ABB RobotStudio station: Process_and_Safety_V2.rsstnx

Station Process_and_Safety_V2 (saved by RobotStudio 23.2.10395.0)
Controller CRB1100_4_47
  mechanical unit ROB_1: CRB1100_4_47__01, 6 joints, base frame (0, 0, 0) mm
Layout (positions relative to the parent item):
  - CRB1100_4_47__01 [mechanism, from %ABB.RobotStudio.Models.CRB1100%\CRB1100_4_47__01.rslib] at (0, 0, 0) mm; joint values [-0.1244, 0.7509, -0.641, 0, 1.4609, -1.6952] (rad or m)
  - My_Mechanism [mechanism] at (0, 0, 0) mm; joint values [0, 0] (rad or m)
      TCP My_Mechanism_1 at (0, 0, 110) mm
      links: L1, L2, L3
  - P001 - Magazine rings [part] at (0, 500, 3) mm, rotated rx 90 ry 0 rz 0 deg, size 68.8 x 79.8 x 194.8 mm
  - P002 - Magazine nuts [part] at (100, 500, 3) mm, rotated rx 90 ry 0 rz 0 deg, size 68.8 x 106.2 x 289.3 mm
  - P004 - Fixture valve body [part] at (400, -50, 19.5) mm, rotated rx 90 ry 0 rz 0 deg, size 55 x 29 x 55 mm
  - P006 - Magazine bodies [part] at (-250, -400, 0) mm, rotated rx 90 ry 0 rz 0 deg, size 68.8 x 305 x 69.5 mm
  - P006a - Magazine bodies support [part] at (-243.75, -400, 85.1) mm, rotated rx 90 ry 0 rz 0 deg, size 40 x 15 x 5 mm
  - P007 - Magazine big nut [part] at (-100, 500, 3) mm, rotated rx 90 ry 0 rz 0 deg, size 68.8 x 91 x 212.5 mm
  - P006a - Magazine bodies support_2 [part] at (-243.75, -400, 145.1) mm, rotated rx 90 ry 0 rz 0 deg, size 40 x 15 x 5 mm
  - P006a - Magazine bodies support_3 [part] at (-243.75, -400, 205.1) mm, rotated rx 90 ry 0 rz 0 deg, size 40 x 15 x 5 mm
  - P006a - Magazine bodies support_4 [part] at (-243.75, -400, 265.1) mm, rotated rx 90 ry 0 rz 0 deg, size 40 x 15 x 5 mm
  - P006a - Magazine bodies support_5 [part] at (-243.75, -400, 25.1) mm, rotated rx 90 ry 0 rz 0 deg, size 40 x 15 x 5 mm
  - A001 - Grijper_2 [part] at (0, 0, 30) mm, rotated rx -90 ry 0 rz 0 deg, size 42 x 60 x 33 mm
  - Part_5 [part] at (0, 0, 30) mm, rotated rx -90 ry 0 rz 0 deg, size 52 x 72 x 22.6 mm
  - Part_6 [part] at (0, 0, 30) mm, rotated rx -90 ry 0 rz 0 deg, size 52 x 72 x 22.6 mm
  - GripperV2 [mechanism] at (89.85, -63.01, 369.8) mm, rotated rx -172.85 ry 3.1 rz -46.9 deg; joint values [0.008, -0.008] (rad or m)
      TCP GripperV2_1 at (0, -80, 0) mm, rotated rx 90 ry 0 rz 0 deg
      links: L1, L2, L3
  - P005 - Grote moer [part] at (-100, 385.14, 20.17) mm, rotated rx 97.62 ry -12.95 rz 59.14 deg, size 34.6 x 16.1 x 30 mm
  - P002 - Moer [part] at (100, 383.67, 26.5) mm, rotated rx 101.36 ry -6.49 rz 29.35 deg, size 24 x 13.5 x 27.7 mm
  - P001 - Sluitring [part] at (0, 381.43, 22.9) mm, rotated rx 103.06 ry 0 rz 0 deg, size 17.4 x 7.9 x 17.5 mm
  - P003 - Verlengstuk [part] at (-203.75, -400, 267.1) mm, rotated rx 0 ry 0 rz 90 deg, size 23.7 x 32 x 23.9 mm
  - P006 - Main Body [part] at (-191.75, -400, 208.6) mm, rotated rx 0 ry 0 rz 90 deg, size 26 x 45.8 x 33.4 mm
  - P002 - Magazine nuts_2 [part] at (200, 500, 3) mm, rotated rx 90 ry 0 rz 0 deg, size 68.8 x 106.2 x 289.3 mm
  - P002 - Moer_2 [part] at (200, 383.67, 26.5) mm, rotated rx -78.64 ry -6.49 rz 29.35 deg, size 24 x 13.5 x 27.7 mm
Attachment: GripperV2 is attached to CRB1100_4_47__01 / Link6
EventTableEntry 2883: ActivationMode=1, Cyclic=false, Group=, Trigger=DO1 2884, Actions=[EventTableActionMechanicalPose 3183], Comment=
EventTableTriggerIO 2884: Operator=0, IOValue=[1], IRC5Controller=? -1, SignalSource=CRB1100_4_47 1186
EventTableTriggerIO 2886: Operator=0, IOValue=[1], IRC5Controller=? -1, SignalSource=CRB1100_4_47 1186
EventTableTriggerIO 2887: Operator=0, IOValue=[1], IRC5Controller=? -1, SignalSource=CRB1100_4_47 1186
EventTableTriggerIO 2888: Operator=0, IOValue=[1], IRC5Controller=? -1, SignalSource=CRB1100_4_47 1186
EventTableTriggerIO 2889: Operator=0, IOValue=[1], IRC5Controller=? -1, SignalSource=CRB1100_4_47 1186
EventTableTriggerIO 2890: Operator=0, IOValue=[1], IRC5Controller=? -1, SignalSource=CRB1100_4_47 1186
EventTableTriggerIO 2891: Operator=0, IOValue=[1], IRC5Controller=? -1, SignalSource=CRB1100_4_47 1186
EventTableTriggerIO 2892: Operator=0, IOValue=[1], IRC5Controller=? -1, SignalSource=CRB1100_4_47 1186
EventTableTriggerIO 2893: Operator=0, IOValue=[1], IRC5Controller=? -1, SignalSource=CRB1100_4_47 1186
EventTableTriggerIO 2894: Operator=0, IOValue=[1], IRC5Controller=? -1, SignalSource=CRB1100_4_47 1186
EventTableTriggerIO 2895: Operator=0, IOValue=[1], IRC5Controller=? -1, SignalSource=CRB1100_4_47 1186
EventTableTriggerIO 2896: Operator=0, IOValue=[1], IRC5Controller=? -1, SignalSource=CRB1100_4_47 1186
EventTableTriggerIO 2897: Operator=0, IOValue=[1], IRC5Controller=? -1, SignalSource=CRB1100_4_47 1186
EventTableTriggerIO 2898: Operator=0, IOValue=[1], IRC5Controller=? -1, SignalSource=CRB1100_4_47 1186
EventTableTriggerIO 2899: Operator=0, IOValue=[1], IRC5Controller=? -1, SignalSource=CRB1100_4_47 1186
EventTableEntry 2900: ActivationMode=1, Cyclic=false, Group=, Trigger=DO2 2901, Actions=[EventTableActionMechanicalPose 3185], Comment=
EventTableTriggerIO 2901: Operator=0, IOValue=[1], IRC5Controller=? -1, SignalSource=CRB1100_4_47 1186
EventTableTriggerIO 2903: Operator=0, IOValue=[1], IRC5Controller=? -1, SignalSource=CRB1100_4_47 1186
EventTableTriggerIO 2904: Operator=0, IOValue=[1], IRC5Controller=? -1, SignalSource=CRB1100_4_47 1186
EventTableTriggerIO 2905: Operator=0, IOValue=[1], IRC5Controller=? -1, SignalSource=CRB1100_4_47 1186
EventTableTriggerIO 2906: Operator=0, IOValue=[1], IRC5Controller=? -1, SignalSource=CRB1100_4_47 1186
EventTableTriggerIO 2907: Operator=0, IOValue=[1], IRC5Controller=? -1, SignalSource=CRB1100_4_47 1186
EventTableTriggerIO 2908: Operator=0, IOValue=[1], IRC5Controller=? -1, SignalSource=CRB1100_4_47 1186
EventTableTriggerIO 2909: Operator=0, IOValue=[1], IRC5Controller=? -1, SignalSource=CRB1100_4_47 1186
EventTableTriggerIO 2910: Operator=0, IOValue=[1], IRC5Controller=? -1, SignalSource=CRB1100_4_47 1186
EventTableTriggerIO 2911: Operator=0, IOValue=[1], IRC5Controller=? -1, SignalSource=CRB1100_4_47 1186
EventTableTriggerIO 2912: Operator=0, IOValue=[1], IRC5Controller=? -1, SignalSource=CRB1100_4_47 1186
EventTableTriggerIO 2913: Operator=0, IOValue=[1], IRC5Controller=? -1, SignalSource=CRB1100_4_47 1186
EventTableTriggerIO 2914: Operator=0, IOValue=[1], IRC5Controller=? -1, SignalSource=CRB1100_4_47 1186
EventTableTriggerIO 2915: Operator=0, IOValue=[1], IRC5Controller=? -1, SignalSource=CRB1100_4_47 1186
EventTableTriggerIO 2916: Operator=0, IOValue=[1], IRC5Controller=? -1, SignalSource=CRB1100_4_47 1186
EventTableTriggerIO 3150: Operator=0, IOValue=[1], IRC5Controller=? -1, SignalSource=CRB1100_4_47 1186
EventTableTriggerIO 3151: Operator=0, IOValue=[1], IRC5Controller=? -1, SignalSource=CRB1100_4_47 1186
EventTableTriggerIO 3152: Operator=0, IOValue=[1], IRC5Controller=? -1, SignalSource=CRB1100_4_47 1186
EventTableTriggerIO 3153: Operator=0, IOValue=[1], IRC5Controller=? -1, SignalSource=CRB1100_4_47 1186
EventTableActionMechanicalPose 3183: VirtualSignal=, Mechanism=GripperV2 3175, ToPoseName=Opened, VirtualSignalValue=[1]
EventTableTriggerIO 3184: Operator=0, IOValue=[1], IRC5Controller=? -1, SignalSource=CRB1100_4_47 1186
EventTableActionMechanicalPose 3185: VirtualSignal=, Mechanism=GripperV2 3175, ToPoseName=Closed, VirtualSignalValue=[1]
EventTableTriggerIO 3186: Operator=0, IOValue=[1], IRC5Controller=? -1, SignalSource=CRB1100_4_47 1186
EventTableEntry 3187: ActivationMode=1, Cyclic=false, Group=, Trigger=EventTableTriggerCollision 3188, Actions=[EventTableActionAttach 3189], Comment=
EventTableTriggerCollision 3188: EventType=0, CollisionSet=CollisionSet_KleineMoer 3195
EventTableActionAttach 3189: MountObject=true, FlangeIndext=0, FindNearest=false, AttachmentParent=GripperV2 3175, AttachmentChild=? -1, Offset=[X=1, Y=0, Z=0, W=0, X=0, Y=1, Z=0, W=0, X=0, Y=0, Z=1, W=0, X=0, Y=0, Z=0, W=1]
EventTableTriggerCollision 3190: EventType=0, CollisionSet=CollisionSet_KleineMoer 3195
EventTableEntry 3191: ActivationMode=1, Cyclic=false, Group=, Trigger=EventTableTriggerCollision 3192, Actions=[EventTableActionDetach 3193], Comment=
EventTableTriggerCollision 3192: EventType=3, CollisionSet=CollisionSet_KleineMoer 3195
EventTableActionDetach 3193: AttachmentParent=GripperV2 3175, AttachmentChild=? -1
EventTableTriggerCollision 3194: EventType=3, CollisionSet=CollisionSet_KleineMoer 3195
Collision set CollisionSet_KleineMoer: P002 - Moer_2 against GripperV2, near miss 0 m
EventTableEntry 3200: ActivationMode=1, Cyclic=false, Group=, Trigger=DO1 3201, Actions=[EventTableActionMechanicalPose 3202], Comment=
EventTableTriggerIO 3201: Operator=0, IOValue=[1], IRC5Controller=? -1, SignalSource=CRB1100_4_47 1186
EventTableActionMechanicalPose 3202: VirtualSignal=, Mechanism=GripperV2 3175, ToPoseName=Opened, VirtualSignalValue=[1]
EventTableTriggerIO 3203: Operator=0, IOValue=[1], IRC5Controller=? -1, SignalSource=CRB1100_4_47 1186
EventTableEntry 3204: ActivationMode=1, Cyclic=false, Group=, Trigger=DO2 3205, Actions=[EventTableActionMechanicalPose 3206], Comment=
EventTableTriggerIO 3205: Operator=0, IOValue=[1], IRC5Controller=? -1, SignalSource=CRB1100_4_47 1186
EventTableActionMechanicalPose 3206: VirtualSignal=, Mechanism=GripperV2 3175, ToPoseName=Closed, VirtualSignalValue=[1]
EventTableTriggerIO 3207: Operator=0, IOValue=[1], IRC5Controller=? -1, SignalSource=CRB1100_4_47 1186
EventTableEntry 3208: ActivationMode=1, Cyclic=false, Group=, Trigger=EventTableTriggerCollision 3209, Actions=[EventTableActionAttach 3210], Comment=
EventTableTriggerCollision 3209: EventType=1, CollisionSet=CollisionSet_KleineMoer 3195
EventTableActionAttach 3210: MountObject=false, FlangeIndext=0, FindNearest=false, AttachmentParent=GripperV2 3175, AttachmentChild=P002 - Moer_2 4207, Offset=[X=1, Y=0, Z=0, W=0, X=0, Y=1, Z=0, W=0, X=0, Y=0, Z=1, W=0, X=0, Y=0, Z=0, W=1]
EventTableTriggerIO 3467: Operator=0, IOValue=[1], IRC5Controller=? -1, SignalSource=CRB1100_4_47 1186
EventTableTriggerIO 3468: Operator=0, IOValue=[1], IRC5Controller=? -1, SignalSource=CRB1100_4_47 1186
EventTableTriggerIO 3469: Operator=0, IOValue=[1], IRC5Controller=? -1, SignalSource=CRB1100_4_47 1186
EventTableTriggerIO 3470: Operator=0, IOValue=[1], IRC5Controller=? -1, SignalSource=CRB1100_4_47 1186
EventTableTriggerIO 3471: Operator=0, IOValue=[1], IRC5Controller=? -1, SignalSource=CRB1100_4_47 1186
EventTableTriggerIO 3472: Operator=0, IOValue=[1], IRC5Controller=? -1, SignalSource=CRB1100_4_47 1186
EventTableTriggerIO 3473: Operator=0, IOValue=[1], IRC5Controller=? -1, SignalSource=CRB1100_4_47 1186
EventTableTriggerIO 3474: Operator=0, IOValue=[1], IRC5Controller=? -1, SignalSource=CRB1100_4_47 1186
EventTableTriggerIO 3475: Operator=0, IOValue=[1], IRC5Controller=? -1, SignalSource=CRB1100_4_47 1186
EventTableTriggerIO 3476: Operator=0, IOValue=[1], IRC5Controller=? -1, SignalSource=CRB1100_4_47 1186
EventTableTriggerCollision 3477: EventType=1, CollisionSet=CollisionSet_KleineMoer 3195
EventTableTriggerCollision 3478: EventType=1, CollisionSet=CollisionSet_KleineMoer 3195
EventTableTriggerCollision 3479: EventType=1, CollisionSet=CollisionSet_KleineMoer 3195
EventTableTriggerCollision 3480: EventType=1, CollisionSet=CollisionSet_KleineMoer 3195
EventTableTriggerCollision 3481: EventType=1, CollisionSet=CollisionSet_KleineMoer 3195
EventTableEntry 3487: ActivationMode=1, Cyclic=false, Group=, Trigger=EventTableTriggerCollision 3488, Actions=[EventTableActionAttach 3489], Comment=
EventTableTriggerCollision 3488: EventType=1, CollisionSet=CollisionSet_Smoring 3493
EventTableActionAttach 3489: MountObject=false, FlangeIndext=0, FindNearest=false, AttachmentParent=GripperV2 3175, AttachmentChild=P003 - Verlengstuk 3845, Offset=[X=1, Y=0, Z=0, W=0, X=0, Y=1, Z=0, W=0, X=0, Y=0, Z=1, W=0, X=0, Y=0, Z=0, W=1]
Collision set CollisionSet_Smoring: P003 - Verlengstuk against GripperV2, near miss 0 m
EventTableTriggerIO 3498: Operator=0, IOValue=[1], IRC5Controller=? -1, SignalSource=CRB1100_4_47 1186
EventTableTriggerIO 3499: Operator=0, IOValue=[1], IRC5Controller=? -1, SignalSource=CRB1100_4_47 1186
EventTableTriggerCollision 3500: EventType=1, CollisionSet=CollisionSet_KleineMoer 3195
EventTableTriggerCollision 3502: EventType=1, CollisionSet=CollisionSet_Smoring 3493
EventTableTriggerIO 3504: Operator=0, IOValue=[1], IRC5Controller=? -1, SignalSource=CRB1100_4_47 1186
EventTableTriggerIO 3505: Operator=0, IOValue=[1], IRC5Controller=? -1, SignalSource=CRB1100_4_47 1186
EventTableTriggerIO 3506: Operator=0, IOValue=[1], IRC5Controller=? -1, SignalSource=CRB1100_4_47 1186
EventTableTriggerIO 3507: Operator=0, IOValue=[1], IRC5Controller=? -1, SignalSource=CRB1100_4_47 1186
EventTableTriggerCollision 3508: EventType=1, CollisionSet=CollisionSet_KleineMoer 3195
EventTableTriggerCollision 3509: EventType=1, CollisionSet=CollisionSet_KleineMoer 3195
EventTableTriggerCollision 3512: EventType=1, CollisionSet=CollisionSet_Smoring 3493
EventTableTriggerCollision 3513: EventType=1, CollisionSet=CollisionSet_Smoring 3493
EventTableTriggerIO 3522: Operator=0, IOValue=[1], IRC5Controller=? -1, SignalSource=CRB1100_4_47 1186
EventTableTriggerIO 3523: Operator=0, IOValue=[1], IRC5Controller=? -1, SignalSource=CRB1100_4_47 1186
EventTableTriggerIO 3524: Operator=0, IOValue=[1], IRC5Controller=? -1, SignalSource=CRB1100_4_47 1186
EventTableTriggerIO 3525: Operator=0, IOValue=[1], IRC5Controller=? -1, SignalSource=CRB1100_4_47 1186
EventTableTriggerIO 3526: Operator=0, IOValue=[1], IRC5Controller=? -1, SignalSource=CRB1100_4_47 1186
EventTableTriggerIO 3527: Operator=0, IOValue=[1], IRC5Controller=? -1, SignalSource=CRB1100_4_47 1186
EventTableTriggerIO 3528: Operator=0, IOValue=[1], IRC5Controller=? -1, SignalSource=CRB1100_4_47 1186
EventTableTriggerIO 3529: Operator=0, IOValue=[1], IRC5Controller=? -1, SignalSource=CRB1100_4_47 1186
EventTableTriggerIO 3530: Operator=0, IOValue=[1], IRC5Controller=? -1, SignalSource=CRB1100_4_47 1186
EventTableTriggerIO 3531: Operator=0, IOValue=[1], IRC5Controller=? -1, SignalSource=CRB1100_4_47 1186
EventTableTriggerCollision 3532: EventType=1, CollisionSet=CollisionSet_KleineMoer 3195
EventTableTriggerCollision 3533: EventType=1, CollisionSet=CollisionSet_KleineMoer 3195
EventTableTriggerCollision 3534: EventType=1, CollisionSet=CollisionSet_KleineMoer 3195
EventTableTriggerCollision 3535: EventType=1, CollisionSet=CollisionSet_KleineMoer 3195
EventTableTriggerCollision 3536: EventType=1, CollisionSet=CollisionSet_KleineMoer 3195
EventTableTriggerCollision 3542: EventType=1, CollisionSet=CollisionSet_Smoring 3493
EventTableTriggerCollision 3543: EventType=1, CollisionSet=CollisionSet_Smoring 3493
EventTableTriggerCollision 3544: EventType=1, CollisionSet=CollisionSet_Smoring 3493
EventTableTriggerCollision 3545: EventType=1, CollisionSet=CollisionSet_Smoring 3493
EventTableTriggerCollision 3546: EventType=1, CollisionSet=CollisionSet_Smoring 3493
EventTableTriggerIO 3622: Operator=0, IOValue=[1], IRC5Controller=? -1, SignalSource=CRB1100_4_47 1186
EventTableTriggerIO 3623: Operator=0, IOValue=[1], IRC5Controller=? -1, SignalSource=CRB1100_4_47 1186
EventTableTriggerIO 3624: Operator=0, IOValue=[1], IRC5Controller=? -1, SignalSource=CRB1100_4_47 1186
EventTableTriggerIO 3625: Operator=0, IOValue=[1], IRC5Controller=? -1, SignalSource=CRB1100_4_47 1186
EventTableTriggerIO 3626: Operator=0, IOValue=[1], IRC5Controller=? -1, SignalSource=CRB1100_4_47 1186
EventTableTriggerIO 3627: Operator=0, IOValue=[1], IRC5Controller=? -1, SignalSource=CRB1100_4_47 1186
EventTableTriggerIO 3628: Operator=0, IOValue=[1], IRC5Controller=? -1, SignalSource=CRB1100_4_47 1186
EventTableTriggerIO 3629: Operator=0, IOValue=[1], IRC5Controller=? -1, SignalSource=CRB1100_4_47 1186
EventTableTriggerIO 3630: Operator=0, IOValue=[1], IRC5Controller=? -1, SignalSource=CRB1100_4_47 1186
EventTableTriggerIO 3631: Operator=0, IOValue=[1], IRC5Controller=? -1, SignalSource=CRB1100_4_47 1186
EventTableTriggerIO 3632: Operator=0, IOValue=[1], IRC5Controller=? -1, SignalSource=CRB1100_4_47 1186
EventTableTriggerIO 3633: Operator=0, IOValue=[1], IRC5Controller=? -1, SignalSource=CRB1100_4_47 1186
EventTableTriggerIO 3634: Operator=0, IOValue=[1], IRC5Controller=? -1, SignalSource=CRB1100_4_47 1186
EventTableTriggerIO 3635: Operator=0, IOValue=[1], IRC5Controller=? -1, SignalSource=CRB1100_4_47 1186
EventTableTriggerIO 3636: Operator=0, IOValue=[1], IRC5Controller=? -1, SignalSource=CRB1100_4_47 1186
EventTableTriggerIO 3637: Operator=0, IOValue=[1], IRC5Controller=? -1, SignalSource=CRB1100_4_47 1186
EventTableTriggerIO 3638: Operator=0, IOValue=[1], IRC5Controller=? -1, SignalSource=CRB1100_4_47 1186
EventTableTriggerIO 3639: Operator=0, IOValue=[1], IRC5Controller=? -1, SignalSource=CRB1100_4_47 1186
EventTableTriggerIO 3640: Operator=0, IOValue=[1], IRC5Controller=? -1, SignalSource=CRB1100_4_47 1186
EventTableTriggerIO 3641: Operator=0, IOValue=[1], IRC5Controller=? -1, SignalSource=CRB1100_4_47 1186
EventTableTriggerIO 3642: Operator=0, IOValue=[1], IRC5Controller=? -1, SignalSource=CRB1100_4_47 1186
EventTableTriggerIO 3643: Operator=0, IOValue=[1], IRC5Controller=? -1, SignalSource=CRB1100_4_47 1186
EventTableTriggerIO 3644: Operator=0, IOValue=[1], IRC5Controller=? -1, SignalSource=CRB1100_4_47 1186
EventTableTriggerIO 3645: Operator=0, IOValue=[1], IRC5Controller=? -1, SignalSource=CRB1100_4_47 1186
EventTableTriggerIO 3646: Operator=0, IOValue=[1], IRC5Controller=? -1, SignalSource=CRB1100_4_47 1186
EventTableTriggerIO 3647: Operator=0, IOValue=[1], IRC5Controller=? -1, SignalSource=CRB1100_4_47 1186
EventTableTriggerCollision 3648: EventType=1, CollisionSet=CollisionSet_KleineMoer 3195
EventTableTriggerCollision 3649: EventType=1, CollisionSet=CollisionSet_KleineMoer 3195
EventTableTriggerCollision 3650: EventType=1, CollisionSet=CollisionSet_KleineMoer 3195
EventTableTriggerCollision 3651: EventType=1, CollisionSet=CollisionSet_KleineMoer 3195
EventTableTriggerCollision 3652: EventType=1, CollisionSet=CollisionSet_KleineMoer 3195
EventTableTriggerCollision 3653: EventType=1, CollisionSet=CollisionSet_KleineMoer 3195
EventTableTriggerCollision 3654: EventType=1, CollisionSet=CollisionSet_KleineMoer 3195
EventTableTriggerCollision 3655: EventType=1, CollisionSet=CollisionSet_KleineMoer 3195
EventTableTriggerCollision 3656: EventType=1, CollisionSet=CollisionSet_KleineMoer 3195
EventTableTriggerCollision 3657: EventType=1, CollisionSet=CollisionSet_KleineMoer 3195
EventTableTriggerCollision 3658: EventType=1, CollisionSet=CollisionSet_KleineMoer 3195
EventTableTriggerCollision 3659: EventType=1, CollisionSet=CollisionSet_KleineMoer 3195
EventTableTriggerCollision 3660: EventType=1, CollisionSet=CollisionSet_KleineMoer 3195
EventTableTriggerCollision 3674: EventType=1, CollisionSet=CollisionSet_Smoring 3493
EventTableTriggerCollision 3675: EventType=1, CollisionSet=CollisionSet_Smoring 3493
EventTableTriggerCollision 3676: EventType=1, CollisionSet=CollisionSet_Smoring 3493
EventTableTriggerCollision 3677: EventType=1, CollisionSet=CollisionSet_Smoring 3493
EventTableTriggerCollision 3678: EventType=1, CollisionSet=CollisionSet_Smoring 3493
EventTableTriggerCollision 3679: EventType=1, CollisionSet=CollisionSet_Smoring 3493
EventTableTriggerCollision 3680: EventType=1, CollisionSet=CollisionSet_Smoring 3493
EventTableTriggerCollision 3681: EventType=1, CollisionSet=CollisionSet_Smoring 3493
EventTableTriggerCollision 3682: EventType=1, CollisionSet=CollisionSet_Smoring 3493
EventTableTriggerCollision 3683: EventType=1, CollisionSet=CollisionSet_Smoring 3493
EventTableTriggerCollision 3684: EventType=1, CollisionSet=CollisionSet_Smoring 3493
EventTableTriggerCollision 3685: EventType=1, CollisionSet=CollisionSet_Smoring 3493
EventTableTriggerCollision 3686: EventType=1, CollisionSet=CollisionSet_Smoring 3493
EventTableTriggerIO 3777: Operator=0, IOValue=[1], IRC5Controller=? -1, SignalSource=CRB1100_4_47 1186
EventTableTriggerIO 3778: Operator=0, IOValue=[1], IRC5Controller=? -1, SignalSource=CRB1100_4_47 1186
EventTableTriggerIO 3779: Operator=0, IOValue=[1], IRC5Controller=? -1, SignalSource=CRB1100_4_47 1186
EventTableTriggerIO 3780: Operator=0, IOValue=[1], IRC5Controller=? -1, SignalSource=CRB1100_4_47 1186
EventTableTriggerIO 3781: Operator=0, IOValue=[1], IRC5Controller=? -1, SignalSource=CRB1100_4_47 1186
EventTableTriggerIO 3782: Operator=0, IOValue=[1], IRC5Controller=? -1, SignalSource=CRB1100_4_47 1186
EventTableTriggerIO 3783: Operator=0, IOValue=[1], IRC5Controller=? -1, SignalSource=CRB1100_4_47 1186
EventTableTriggerIO 3784: Operator=0, IOValue=[1], IRC5Controller=? -1, SignalSource=CRB1100_4_47 1186
EventTableTriggerIO 3785: Operator=0, IOValue=[1], IRC5Controller=? -1, SignalSource=CRB1100_4_47 1186
EventTableTriggerIO 3786: Operator=0, IOValue=[1], IRC5Controller=? -1, SignalSource=CRB1100_4_47 1186
EventTableTriggerIO 3787: Operator=0, IOValue=[1], IRC5Controller=? -1, SignalSource=CRB1100_4_47 1186
EventTableTriggerIO 3788: Operator=0, IOValue=[1], IRC5Controller=? -1, SignalSource=CRB1100_4_47 1186
EventTableTriggerCollision 3789: EventType=1, CollisionSet=CollisionSet_KleineMoer 3195
EventTableTriggerCollision 3790: EventType=1, CollisionSet=CollisionSet_KleineMoer 3195
EventTableTriggerCollision 3791: EventType=1, CollisionSet=CollisionSet_KleineMoer 3195
EventTableTriggerCollision 3792: EventType=1, CollisionSet=CollisionSet_KleineMoer 3195
EventTableTriggerCollision 3793: EventType=3, CollisionSet=CollisionSet_KleineMoer 3195
EventTableTriggerCollision 3794: EventType=0, CollisionSet=CollisionSet_KleineMoer 3195
EventTableTriggerCollision 3795: EventType=1, CollisionSet=CollisionSet_Smoring 3493
EventTableTriggerCollision 3796: EventType=1, CollisionSet=CollisionSet_Smoring 3493
EventTableTriggerCollision 3797: EventType=1, CollisionSet=CollisionSet_Smoring 3493
EventTableTriggerCollision 3798: EventType=1, CollisionSet=CollisionSet_Smoring 3493
EventTableTriggerCollision 3799: EventType=3, CollisionSet=CollisionSet_Smoring 3493
EventTableTriggerCollision 3800: EventType=0, CollisionSet=CollisionSet_Smoring 3493
EventTableEntry 3801: ActivationMode=1, Cyclic=false, Group=, Trigger=EventTableTriggerCollision 3802, Actions=[EventTableActionAttach 3803], Comment=
EventTableTriggerCollision 3802: EventType=1, CollisionSet=CollisionSet_KleineMoer2 3804
EventTableActionAttach 3803: MountObject=false, FlangeIndext=0, FindNearest=false, AttachmentParent=P004 - Fixture valve body 2400, AttachmentChild=P002 - Moer_2 4207, Offset=[X=1, Y=0, Z=0, W=0, X=0, Y=1, Z=0, W=0, X=0, Y=0, Z=1, W=0, X=0, Y=0, Z=0, W=1]
Collision set CollisionSet_KleineMoer2: P002 - Moer_2 against P004 - Fixture valve body, near miss 0 m
Collision set CollisionSet_Smoring2: P003 - Verlengstuk against P002 - Moer_2, near miss 0 m
EventTableTriggerIO 3812: Operator=0, IOValue=[1], IRC5Controller=? -1, SignalSource=CRB1100_4_47 1186
EventTableTriggerIO 3813: Operator=0, IOValue=[1], IRC5Controller=? -1, SignalSource=CRB1100_4_47 1186
EventTableTriggerIO 3814: Operator=0, IOValue=[1], IRC5Controller=? -1, SignalSource=CRB1100_4_47 1186
EventTableTriggerIO 3816: Operator=0, IOValue=[1], IRC5Controller=? -1, SignalSource=CRB1100_4_47 1186
EventTableTriggerIO 3817: Operator=0, IOValue=[1], IRC5Controller=? -1, SignalSource=CRB1100_4_47 1186
EventTableTriggerIO 3818: Operator=0, IOValue=[1], IRC5Controller=? -1, SignalSource=CRB1100_4_47 1186
EventTableTriggerCollision 3820: EventType=1, CollisionSet=CollisionSet_KleineMoer 3195
EventTableTriggerCollision 3821: EventType=1, CollisionSet=CollisionSet_KleineMoer 3195
EventTableTriggerCollision 3822: EventType=1, CollisionSet=CollisionSet_KleineMoer 3195
EventTableTriggerCollision 3824: EventType=1, CollisionSet=CollisionSet_Smoring 3493
EventTableTriggerCollision 3825: EventType=1, CollisionSet=CollisionSet_Smoring 3493
EventTableTriggerCollision 3826: EventType=1, CollisionSet=CollisionSet_Smoring 3493
EventTableTriggerCollision 3828: EventType=1, CollisionSet=CollisionSet_KleineMoer2 3804
EventTableTriggerCollision 3829: EventType=1, CollisionSet=CollisionSet_KleineMoer2 3804
EventTableTriggerCollision 3830: EventType=1, CollisionSet=CollisionSet_KleineMoer2 3804
EventTableEntry 3832: ActivationMode=1, Cyclic=false, Group=, Trigger=EventTableTriggerCollision 3833, Actions=[EventTableActionAttach 3834], Comment=
EventTableTriggerCollision 3833: EventType=1, CollisionSet=CollisionSet_Smoring2 3805
EventTableActionAttach 3834: MountObject=false, FlangeIndext=0, FindNearest=false, AttachmentParent=P002 - Moer_2 4207, AttachmentChild=P003 - Verlengstuk 3845, Offset=[X=1, Y=0, Z=0, W=0, X=0, Y=1, Z=0, W=0, X=0, Y=0, Z=1, W=0, X=0, Y=0, Z=0, W=1]
EventTableTriggerCollision 3835: EventType=1, CollisionSet=CollisionSet_Smoring2 3805
EventTableTriggerCollision 3836: EventType=1, CollisionSet=CollisionSet_Smoring2 3805
EventTableTriggerCollision 3837: EventType=1, CollisionSet=CollisionSet_Smoring2 3805
EventTableTriggerIO 3848: Operator=0, IOValue=[1], IRC5Controller=? -1, SignalSource=CRB1100_4_47 1186
EventTableTriggerIO 3849: Operator=0, IOValue=[1], IRC5Controller=? -1, SignalSource=CRB1100_4_47 1186
EventTableTriggerIO 3850: Operator=0, IOValue=[1], IRC5Controller=? -1, SignalSource=CRB1100_4_47 1186
EventTableTriggerIO 3851: Operator=0, IOValue=[1], IRC5Controller=? -1, SignalSource=CRB1100_4_47 1186
EventTableTriggerIO 3852: Operator=0, IOValue=[1], IRC5Controller=? -1, SignalSource=CRB1100_4_47 1186
EventTableTriggerIO 3853: Operator=0, IOValue=[1], IRC5Controller=? -1, SignalSource=CRB1100_4_47 1186
EventTableTriggerIO 3854: Operator=0, IOValue=[1], IRC5Controller=? -1, SignalSource=CRB1100_4_47 1186
EventTableTriggerIO 3855: Operator=0, IOValue=[1], IRC5Controller=? -1, SignalSource=CRB1100_4_47 1186
EventTableTriggerCollision 3856: EventType=1, CollisionSet=CollisionSet_KleineMoer 3195
EventTableTriggerCollision 3857: EventType=1, CollisionSet=CollisionSet_KleineMoer 3195
EventTableTriggerCollision 3858: EventType=1, CollisionSet=CollisionSet_KleineMoer 3195
EventTableTriggerCollision 3859: EventType=1, CollisionSet=CollisionSet_KleineMoer 3195
EventTableTriggerCollision 3860: EventType=1, CollisionSet=CollisionSet_Smoring 3493
EventTableTriggerCollision 3861: EventType=1, CollisionSet=CollisionSet_Smoring 3493
EventTableTriggerCollision 3862: EventType=1, CollisionSet=CollisionSet_Smoring 3493
EventTableTriggerCollision 3863: EventType=1, CollisionSet=CollisionSet_Smoring 3493
EventTableTriggerCollision 3864: EventType=1, CollisionSet=CollisionSet_KleineMoer2 3804
EventTableTriggerCollision 3865: EventType=1, CollisionSet=CollisionSet_KleineMoer2 3804
EventTableTriggerCollision 3866: EventType=1, CollisionSet=CollisionSet_KleineMoer2 3804
EventTableTriggerCollision 3867: EventType=1, CollisionSet=CollisionSet_KleineMoer2 3804
EventTableTriggerCollision 3868: EventType=1, CollisionSet=CollisionSet_Smoring2 3805
EventTableTriggerCollision 3869: EventType=1, CollisionSet=CollisionSet_Smoring2 3805
EventTableTriggerCollision 3870: EventType=1, CollisionSet=CollisionSet_Smoring2 3805
EventTableTriggerCollision 3871: EventType=1, CollisionSet=CollisionSet_Smoring2 3805
EventTableTriggerIO 4069: Operator=0, IOValue=[1], IRC5Controller=? -1, SignalSource=CRB1100_4_47 1186
EventTableTriggerIO 4070: Operator=0, IOValue=[1], IRC5Controller=? -1, SignalSource=CRB1100_4_47 1186
EventTableTriggerIO 4071: Operator=0, IOValue=[1], IRC5Controller=? -1, SignalSource=CRB1100_4_47 1186
EventTableTriggerIO 4072: Operator=0, IOValue=[1], IRC5Controller=? -1, SignalSource=CRB1100_4_47 1186
EventTableTriggerCollision 4073: EventType=1, CollisionSet=CollisionSet_KleineMoer 3195
EventTableTriggerCollision 4074: EventType=1, CollisionSet=CollisionSet_KleineMoer 3195
EventTableTriggerCollision 4075: EventType=1, CollisionSet=CollisionSet_Smoring 3493
EventTableTriggerCollision 4076: EventType=1, CollisionSet=CollisionSet_Smoring 3493
EventTableTriggerCollision 4077: EventType=1, CollisionSet=CollisionSet_KleineMoer2 3804
EventTableTriggerCollision 4078: EventType=1, CollisionSet=CollisionSet_KleineMoer2 3804
EventTableTriggerCollision 4079: EventType=1, CollisionSet=CollisionSet_Smoring2 3805
EventTableTriggerCollision 4080: EventType=1, CollisionSet=CollisionSet_Smoring2 3805
EventTableTriggerIO 4081: Operator=0, IOValue=[1], IRC5Controller=? -1, SignalSource=CRB1100_4_47 1186
EventTableTriggerIO 4082: Operator=0, IOValue=[1], IRC5Controller=? -1, SignalSource=CRB1100_4_47 1186
EventTableTriggerIO 4083: Operator=0, IOValue=[1], IRC5Controller=? -1, SignalSource=CRB1100_4_47 1186
EventTableTriggerIO 4084: Operator=0, IOValue=[1], IRC5Controller=? -1, SignalSource=CRB1100_4_47 1186
EventTableTriggerIO 4085: Operator=0, IOValue=[1], IRC5Controller=? -1, SignalSource=CRB1100_4_47 1186
EventTableTriggerIO 4086: Operator=0, IOValue=[1], IRC5Controller=? -1, SignalSource=CRB1100_4_47 1186
EventTableTriggerCollision 4087: EventType=1, CollisionSet=CollisionSet_KleineMoer 3195
EventTableTriggerCollision 4088: EventType=1, CollisionSet=CollisionSet_KleineMoer 3195
EventTableTriggerCollision 4089: EventType=1, CollisionSet=CollisionSet_KleineMoer 3195
EventTableTriggerCollision 4090: EventType=1, CollisionSet=CollisionSet_Smoring 3493
EventTableTriggerCollision 4091: EventType=1, CollisionSet=CollisionSet_Smoring 3493
EventTableTriggerCollision 4092: EventType=1, CollisionSet=CollisionSet_Smoring 3493
EventTableTriggerCollision 4093: EventType=1, CollisionSet=CollisionSet_KleineMoer2 3804
EventTableTriggerCollision 4094: EventType=1, CollisionSet=CollisionSet_KleineMoer2 3804
EventTableTriggerCollision 4095: EventType=1, CollisionSet=CollisionSet_KleineMoer2 3804
EventTableTriggerCollision 4096: EventType=1, CollisionSet=CollisionSet_Smoring2 3805
EventTableTriggerCollision 4097: EventType=1, CollisionSet=CollisionSet_Smoring2 3805
EventTableTriggerCollision 4098: EventType=1, CollisionSet=CollisionSet_Smoring2 3805
EventTableTriggerIO 4100: Operator=0, IOValue=[1], IRC5Controller=? -1, SignalSource=CRB1100_4_47 1186
EventTableTriggerIO 4101: Operator=0, IOValue=[1], IRC5Controller=? -1, SignalSource=CRB1100_4_47 1186
EventTableTriggerIO 4102: Operator=0, IOValue=[1], IRC5Controller=? -1, SignalSource=CRB1100_4_47 1186
EventTableTriggerIO 4103: Operator=0, IOValue=[1], IRC5Controller=? -1, SignalSource=CRB1100_4_47 1186
EventTableTriggerIO 4104: Operator=0, IOValue=[1], IRC5Controller=? -1, SignalSource=CRB1100_4_47 1186
EventTableTriggerIO 4105: Operator=0, IOValue=[1], IRC5Controller=? -1, SignalSource=CRB1100_4_47 1186
EventTableTriggerCollision 4106: EventType=1, CollisionSet=CollisionSet_KleineMoer 3195
EventTableTriggerCollision 4107: EventType=1, CollisionSet=CollisionSet_KleineMoer 3195
EventTableTriggerCollision 4108: EventType=1, CollisionSet=CollisionSet_KleineMoer 3195
EventTableTriggerCollision 4109: EventType=1, CollisionSet=CollisionSet_Smoring 3493
EventTableTriggerCollision 4110: EventType=1, CollisionSet=CollisionSet_Smoring 3493
EventTableTriggerCollision 4111: EventType=1, CollisionSet=CollisionSet_Smoring 3493
EventTableTriggerCollision 4112: EventType=1, CollisionSet=CollisionSet_KleineMoer2 3804
EventTableTriggerCollision 4113: EventType=1, CollisionSet=CollisionSet_KleineMoer2 3804
EventTableTriggerCollision 4114: EventType=1, CollisionSet=CollisionSet_KleineMoer2 3804
EventTableTriggerCollision 4115: EventType=1, CollisionSet=CollisionSet_Smoring2 3805
EventTableTriggerCollision 4116: EventType=1, CollisionSet=CollisionSet_Smoring2 3805
EventTableTriggerCollision 4117: EventType=1, CollisionSet=CollisionSet_Smoring2 3805
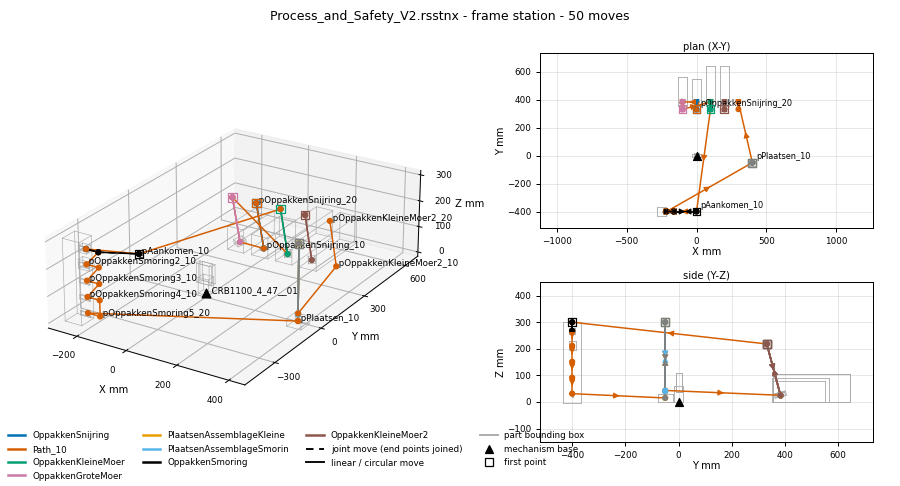
[picture p0: tool path of Process_and_Safety_V2.rsstnx in frame station, 50 of 50 moves have a stored position in this frame; points joined in program order, loops and branches not executed]
Targets, tools, work objects and paths stored in the station, written as RAPID:
! task T_ROB1
MODULE CalibData
  PERS tooldata Gripper_1:=[TRUE,[[200,-78.998,0],[0.707106781,0.707106781,0,0]],[1,[0,35,0],[1,0,0,0],0,0,0]];
  PERS tooldata My_Mechanism_1:=[TRUE,[[0,0,110],[1,0,0,0]],[1,[0,0,60],[1,0,0,0],0,0,0]];
  PERS wobjdata OpslagGroteMoer:=[FALSE,TRUE,"",[[-118.446955384,558.318847229,91.427680557],[0.130523756,-0.99144446,-0.001184707,-0.00016626]],[[0,0,0],[1,0,0,0]]];
  PERS wobjdata OpslagSnijring:=[FALSE,TRUE,"",[[-11.83,545.855,80.324],[0.13052697,-0.991444759,0,0]],[[0,0,0],[1,0,0,0]]];
  PERS wobjdata OpslagKleineMoer:=[FALSE,TRUE,"",[[84.95,640.257,106.654],[0.130526202,-0.99144486,0,0]],[[0,0,0],[1,0,0,0]]];
  PERS wobjdata AssemblageKlep:=[FALSE,TRUE,"",[[382.5,-67.5,10],[1,0,0,0]],[[0,0,0],[1,0,0,0]]];
  PERS wobjdata OpslagSmoring:=[FALSE,TRUE,"",[[41.25,-408.75,301.5],[1,0,0,0]],[[-300,0,0],[1,0,0,0]]];
  PERS tooldata GripperV2_1:=[TRUE,[[0,0,110],[1,0,0,0]],[1,[0,0,50],[1,0,0,0],0,0,0]];
  TASK PERS wobjdata OpslagKleineMoer2:=[FALSE,TRUE,"",[[184.95,640.26,106.65],[0.130526192,-0.991444861,0,0]],[[0,0,0],[1,0,0,0]]];
ENDMODULE

! task T_ROB1
MODULE Module1
  CONST robtarget pOppakkenSmoring1_10:=[[45,8.75,-34.4],[0.5,0.5,-0.5,-0.5],[-2,-2,-2,0],[9E+09,9E+09,9E+09,9E+09,9E+09,9E+09]];
  CONST robtarget pOppakkenSmoring2_10:=[[45,8.75,-90.4],[0.5,0.5,-0.5,-0.5],[-2,-2,-2,0],[9E+09,9E+09,9E+09,9E+09,9E+09,9E+09]];
  CONST robtarget pOppakkenSmoring3_10:=[[45,8.75,-150.4],[0.5,0.5,-0.5,-0.5],[-2,-2,-2,0],[9E+09,9E+09,9E+09,9E+09,9E+09,9E+09]];
  CONST robtarget pOppakkenSmoring4_10:=[[45,8.75,-210.4],[0.5,0.5,-0.5,-0.5],[-2,-2,-2,0],[9E+09,9E+09,9E+09,9E+09,9E+09,9E+09]];
  CONST robtarget pOppakkenSmoring5_10:=[[45,8.75,-270.4],[0.5,0.5,-0.5,-0.5],[0,0,0,0],[9E+09,9E+09,9E+09,9E+09,9E+09,9E+09]];
  CONST robtarget pOppakkenSmoring1_20:=[[95,8.75,-34.4],[0.5,0.5,-0.5,-0.5],[-1,-1,-2,0],[9E+09,9E+09,9E+09,9E+09,9E+09,9E+09]];
  CONST robtarget pOppakkenSmoring2_20:=[[95,8.75,-90.4],[0.5,0.5,-0.5,-0.5],[-1,-1,-2,0],[9E+09,9E+09,9E+09,9E+09,9E+09,9E+09]];
  CONST robtarget pOppakkenSmoring3_20:=[[95,8.75,-150.4],[0.5,0.5,-0.5,-0.5],[-1,-1,-2,0],[9E+09,9E+09,9E+09,9E+09,9E+09,9E+09]];
  CONST robtarget pOppakkenSmoring4_20:=[[95,8.75,-210.4],[0.5,0.5,-0.5,-0.5],[-1,-1,-2,0],[9E+09,9E+09,9E+09,9E+09,9E+09,9E+09]];
  CONST robtarget pOppakkenSmoring5_20:=[[95,8.75,-270.4],[0.5,0.5,-0.5,-0.5],[0,0,0,0],[9E+09,9E+09,9E+09,9E+09,9E+09,9E+09]];
  CONST robtarget pAankomen_10:=[[258.75,8.75,-1.5],[0,-0.707106781,0.707106781,0],[-1,0,-2,0],[9E+09,9E+09,9E+09,9E+09,9E+09,9E+09]];
  CONST robtarget pPlaatsen_10:=[[17.5,17.5,5],[0,0,1,0],[-1,0,1,0],[9E+09,9E+09,9E+09,9E+09,9E+09,9E+09]];
  CONST robtarget pPlaatsenKleineMoer_20:=[[17.5,17.5,290],[0,-0.707106781,0.707106781,0],[0,0,0,0],[9E+09,9E+09,9E+09,9E+09,9E+09,9E+09]];
  CONST robtarget pOppakkenKleineMoer_10:=[[15.05,268.809153632,12.497268931],[1,-0.000000009,0,0],[0,0,-2,0],[9E+09,9E+09,9E+09,9E+09,9E+09,9E+09]];
  CONST robtarget pOppakkenKleineMoer_20:=[[15.05,268.809150032,-187.502731069],[1,-0.000000009,0,0],[0,0,-2,0],[9E+09,9E+09,9E+09,9E+09,9E+09,9E+09]];
  CONST robtarget pOppakkenSnijring_10:=[[11.83,170.809139248,13.497214734],[1,-0.000000784,0,0],[1,0,-2,0],[9E+09,9E+09,9E+09,9E+09,9E+09,9E+09]];
  CONST robtarget pOppakkenGroteMoer_10:=[[18.00216669,185.765627355,18.998183197],[0.999999284,0.000002364,-0.000010202,0.001196273],[1,-1,-1,0],[9E+09,9E+09,9E+09,9E+09,9E+09,9E+09]];
  CONST robtarget pOppakkenSnijring_20:=[[11.83,170.808822668,-188.502785265],[1,-0.000000784,0,0],[1,0,-2,0],[9E+09,9E+09,9E+09,9E+09,9E+09,9E+09]];
  CONST robtarget pOppakkenGroteMoer_20:=[[18.006246487,185.766577781,-181.00181676],[0.999999284,0.000002364,-0.000010202,0.001196273],[1,-1,-1,0],[9E+09,9E+09,9E+09,9E+09,9E+09,9E+09]];
  CONST robtarget pPlaatsenSmoring20:=[[17.499997701,17.500002439,33.319985801],[-0.000000013,0.981307099,-0.192448378,-0.000000021],[-1,-1,-2,0],[9E+09,9E+09,9E+09,9E+09,9E+09,9E+09]];
  CONST robtarget pPlaatsenSmoring10:=[[17.500002738,17.499999768,28.999977289],[-0.000000004,0.91420252,0.405257638,0.000000012],[-1,0,1,0],[9E+09,9E+09,9E+09,9E+09,9E+09,9E+09]];
  CONST robtarget pOppakkenKleineMoer2_10:=[[115.05,268.809153632,12.497268931],[1,-0.000000009,0,0],[0,0,-2,0],[9E+09,9E+09,9E+09,9E+09,9E+09,9E+09]];
  CONST robtarget pOppakkenKleineMoer2_20:=[[115.05,268.809150032,-187.502731069],[1,-0.000000009,0,0],[0,0,-2,0],[9E+09,9E+09,9E+09,9E+09,9E+09,9E+09]];
  PROC OppakkenSnijring()
    MoveJDO pOppakkenSnijring_20,V500,fine,My_Mechanism_1\WObj:=OpslagSnijring,DO2,0;
    SetDO DO1,1;
    MoveL pOppakkenSnijring_10,V500,fine,My_Mechanism_1\WObj:=OpslagSnijring;
    SetDO DO1,0;
    SetDO DO2,1;
    WaitTime 0.5;
    MoveL pOppakkenSnijring_20,V500,fine,My_Mechanism_1\WObj:=OpslagSnijring;
  ENDPROC
  PROC Path_10()
    MoveL pOppakkenSnijring_20,v1000,z100,My_Mechanism_1\WObj:=OpslagSnijring;
    MoveL pOppakkenSnijring_10,v1000,z100,My_Mechanism_1\WObj:=OpslagSnijring;
    MoveL pOppakkenGroteMoer_10,v1000,z100,My_Mechanism_1\WObj:=OpslagGroteMoer;
    MoveL pOppakkenGroteMoer_20,v1000,z100,My_Mechanism_1\WObj:=OpslagGroteMoer;
    MoveL pOppakkenKleineMoer_10,v1000,z100,My_Mechanism_1\WObj:=OpslagKleineMoer;
    MoveL pOppakkenKleineMoer_20,v1000,z100,My_Mechanism_1\WObj:=OpslagKleineMoer;
    MoveL pAankomen_10,v1000,z100,My_Mechanism_1\WObj:=OpslagSmoring;
    MoveL pOppakkenSmoring1_10,v1000,z100,My_Mechanism_1\WObj:=OpslagSmoring;
    MoveL pOppakkenSmoring1_20,v1000,z100,My_Mechanism_1\WObj:=OpslagSmoring;
    MoveL pOppakkenSmoring2_10,v1000,z100,My_Mechanism_1\WObj:=OpslagSmoring;
    MoveL pOppakkenSmoring2_20,v1000,z100,My_Mechanism_1\WObj:=OpslagSmoring;
    MoveL pOppakkenSmoring3_10,v1000,z100,My_Mechanism_1\WObj:=OpslagSmoring;
    MoveL pOppakkenSmoring3_20,v1000,z100,My_Mechanism_1\WObj:=OpslagSmoring;
    MoveL pOppakkenSmoring4_10,v1000,z100,My_Mechanism_1\WObj:=OpslagSmoring;
    MoveL pOppakkenSmoring4_20,v1000,z100,My_Mechanism_1\WObj:=OpslagSmoring;
    MoveL pOppakkenSmoring5_20,v1000,z100,My_Mechanism_1\WObj:=OpslagSmoring;
    MoveL pOppakkenSmoring5_10,v1000,z100,My_Mechanism_1\WObj:=OpslagSmoring;
    MoveL pPlaatsen_10,v1000,z100,My_Mechanism_1\WObj:=AssemblageKlep;
    MoveL pPlaatsenKleineMoer_20,v1000,z100,My_Mechanism_1\WObj:=AssemblageKlep;
    MoveL pPlaatsenSmoring10,v1000,z100,GripperV2_1\WObj:=AssemblageKlep;
    MoveL pPlaatsenSmoring20,v1000,z100,GripperV2_1\WObj:=AssemblageKlep;
    MoveL pOppakkenKleineMoer2_10,v1000,z100,GripperV2_1\WObj:=OpslagKleineMoer2;
    MoveL pOppakkenKleineMoer2_20,v1000,z100,GripperV2_1\WObj:=OpslagKleineMoer2;
  ENDPROC
  PROC OppakkenKleineMoer()
    MoveJDO pOppakkenKleineMoer_20,V500,fine,My_Mechanism_1\WObj:=OpslagKleineMoer,DO2,0;
    SetDO DO1,1;
    MoveL pOppakkenKleineMoer_10,V500,fine,My_Mechanism_1\WObj:=OpslagKleineMoer;
    SetDO DO1,0;
    SetDO DO2,1;
    WaitTime 0.5;
    MoveL pOppakkenKleineMoer_20,V500,fine,My_Mechanism_1\WObj:=OpslagKleineMoer;
  ENDPROC
  PROC OppakkenGroteMoer()
    MoveJDO pOppakkenGroteMoer_20,V500,fine,My_Mechanism_1\WObj:=OpslagGroteMoer,DO2,0;
    SetDO DO1,1;
    MoveL pOppakkenGroteMoer_10,V500,fine,My_Mechanism_1\WObj:=OpslagGroteMoer;
    SetDO DO1,0;
    SetDO DO2,1;
    WaitTime 0.5;
    MoveL pOppakkenGroteMoer_20,V500,fine,My_Mechanism_1\WObj:=OpslagGroteMoer;
  ENDPROC
  PROC MainProtocol()
    OppakkenKleineMoer2;
    PlaatsenAssemblageKleineMoer2;
    OppakkenSmoring;
    PlaatsenAssemblageSmoring;
  ENDPROC
  PROC PlaatsenAssemblageKleineMoer()
    MoveJ pPlaatsenKleineMoer_20,V200,fine,My_Mechanism_1\WObj:=AssemblageKlep;
    MoveL pPlaatsen_10,V200,fine,My_Mechanism_1\WObj:=AssemblageKlep;
    WaitTime 0.5;
    SetDO DO2,0;
    SetDO DO1,1;
    WaitTime 0.5;
    MoveL pPlaatsenKleineMoer_20,V200,fine,My_Mechanism_1\WObj:=AssemblageKlep;
  ENDPROC
  PROC PlaatsenAssemblageSmoring()
    MoveJ pPlaatsenKleineMoer_20,V200,fine,My_Mechanism_1\WObj:=AssemblageKlep;
    MoveL pPlaatsenSmoring20,V200,fine,My_Mechanism_1\WObj:=AssemblageKlep;
    MoveJ pPlaatsenSmoring10,V200,fine,My_Mechanism_1\WObj:=AssemblageKlep;
    SetDO DO2,0;
    SetDO DO1,1;
    WaitTime 0.5;
    MoveL pPlaatsenKleineMoer_20,V200,fine,My_Mechanism_1\WObj:=AssemblageKlep;
    WaitTime 0.5;
  ENDPROC
  PROC OppakkenSmoring()
    MoveJ pAankomen_10,V200,fine,My_Mechanism_1\WObj:=OpslagSmoring;
    MoveLDO pOppakkenSmoring1_20,V200,fine,My_Mechanism_1\WObj:=OpslagSmoring,DO2,0;
    SetDO DO1,1;
    MoveL pOppakkenSmoring1_10,V200,fine,My_Mechanism_1\WObj:=OpslagSmoring;
    SetDO DO1,0;
    SetDO DO2,1;
    WaitTime 0.5;
    MoveL pOppakkenSmoring1_20,V200,fine,My_Mechanism_1\WObj:=OpslagSmoring;
    MoveJ pAankomen_10,V200,fine,My_Mechanism_1\WObj:=OpslagSmoring;
  ENDPROC
  PROC PlaatsenSmoring()
  ENDPROC
  PROC OppakkenKleineMoer2()
    MoveJDO pOppakkenKleineMoer2_20,V500,fine,My_Mechanism_1\WObj:=OpslagKleineMoer,DO2,0;
    SetDO DO1,1;
    MoveL pOppakkenKleineMoer2_10,V500,fine,My_Mechanism_1\WObj:=OpslagKleineMoer;
    SetDO DO1,0;
    SetDO DO2,1;
    WaitTime 0.5;
    MoveL pOppakkenKleineMoer2_20,V500,fine,My_Mechanism_1\WObj:=OpslagKleineMoer;
  ENDPROC
  PROC PlaatsenAssemblageKleineMoer2()
    MoveJ pPlaatsenKleineMoer_20,V200,fine,My_Mechanism_1\WObj:=AssemblageKlep;
    MoveL pPlaatsen_10,V200,fine,My_Mechanism_1\WObj:=AssemblageKlep;
    WaitTime 0.5;
    SetDO DO2,0;
    SetDO DO1,1;
    WaitTime 0.5;
    MoveL pPlaatsenKleineMoer_20,V200,fine,My_Mechanism_1\WObj:=AssemblageKlep;
  ENDPROC
ENDMODULE

